{attribute 'qualified_only'}
{attribute 'strict'}
TYPE E_DBStnLED :
(
	PurgeButton	:= 5
);
END_TYPE

(* stored: Version 1.1.0.1, ProductVersion 3.1.4022.18
   DUT E_DBStnLED: Id {86294486-7412-4bb9-b783-f69a0fdc46bf} *)
